FUNCTION_BLOCK PUBLIC PAEJamSensor EXTENDS PAESensorDigital
VAR_INPUT
END_VAR
VAR_OUTPUT
END_VAR
VAR
END_VAR

END_FUNCTION_BLOCK

(* stored: Version 1.1.0.1, ProductVersion 3.1.4020.6
   POU PAEJamSensor: Id {a37adc90-bc67-4c1d-9c58-f4cbef4912a5}, SpecialFunc None *)
